PROGRAM MAIN
VAR
	heartbeat: INT;
END_VAR

heartbeat := heartbeat + 1;

END_PROGRAM

(* stored: Version 1.1.0.1, ProductVersion 3.1.4024.0
   POU MAIN: Id {4d39b111-49e2-4740-8f14-2e7af4926307}, SpecialFunc None *)
